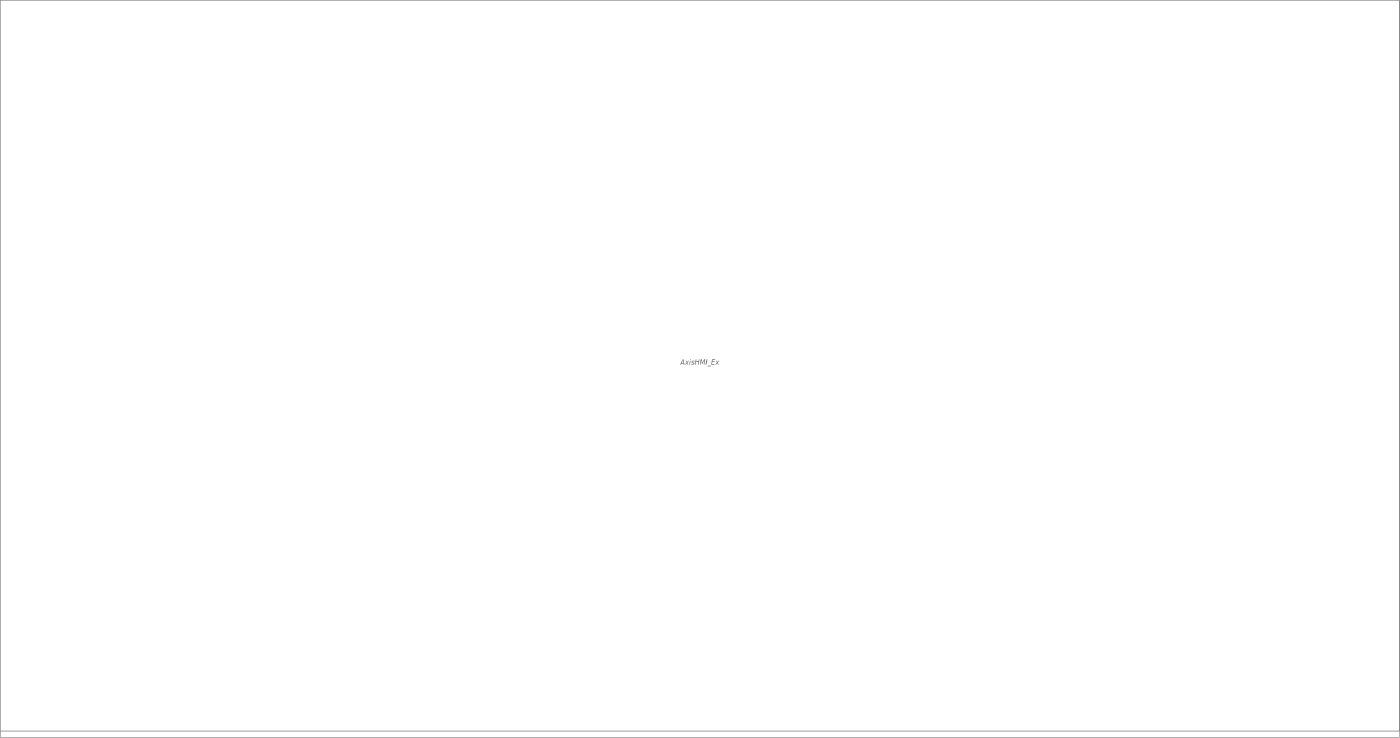
VISUALIZATION visu_working1  // 2048x1080
    TabControl (0,-10 2048x1080)
        shows AxisHMI_Ex(stAxisHMI := GVL.fb_working1.st_mcAxis_lift, mcAxis := GVL.fb_working1.mcAxis_lift, xError := GVL.fb_working1.mcAxis_lift.xError)
        shows AxisHMI_Ex(stAxisHMI := GVL.fb_working1.st_mcAxis_bag, mcAxis := GVL.fb_working1.mcAxis_bag, xError := GVL.fb_working1.mcAxis_bag.xError)
        shows v_io_working1()
        shows AxisHMI_Ex(stAxisHMI := GVL.fb_working.st_mcAxis_vacuun[0], mcAxis := GVL.fb_working.mcAxis_vacuun[0], xError := GVL.fb_working.mcAxis_vacuun[0].xError)
        shows AxisHMI_Ex(stAxisHMI := GVL.fb_working.st_mcAxis_vacuun[1], mcAxis := GVL.fb_working.mcAxis_vacuun[1], xError := GVL.fb_working.mcAxis_vacuun[1].xError)
        shows AxisHMI_Ex(stAxisHMI := GVL.fb_working.st_mcAxis_bagOpen[0], mcAxis := GVL.fb_working.mcAxis_bagOpen[0], xError := GVL.fb_working.mcAxis_bagOpen[0].xError)
        shows AxisHMI_Ex(stAxisHMI := GVL.fb_working.st_mcAxis_bagOpen[1], mcAxis := GVL.fb_working.mcAxis_bagOpen[1], xError := GVL.fb_working.mcAxis_bagOpen[1].xError)
        shows AxisHMI_Ex(stAxisHMI := GVL.fb_working.st_mcAxis_bagOpen[2], mcAxis := GVL.fb_working.mcAxis_bagOpen[2], xError := GVL.fb_working.mcAxis_bagOpen[2].xError)
        shows AxisHMI_Ex(stAxisHMI := GVL.fb_working.st_mcAxis_bagOpen[3], mcAxis := GVL.fb_working.mcAxis_bagOpen[3], xError := GVL.fb_working.mcAxis_bagOpen[3].xError)
        [0]: TabTitle=Lift
        [1]: TabTitle=BagOpen
        [3]: TabTitle=Axis_vacuun_0
        [4]: TabTitle=Axis_vacuun_1
        [5]: TabTitle=Axis_bagOpen_0
        [6]: TabTitle=Axis_bagOpen_1
        [7]: TabTitle=Axis_bagOpen_2
        [8]: TabTitle=Axis_bagOpen_3
        p2837713833: gantrybase.mcAxis[EN_Axis.Z].sAxisName
END_VISUALIZATION

(* stored: Version 1.1.0.1, ProductVersion 3.1.4024.12
   Visu visu_working1: Id {4237067d-ba12-473e-bb87-3d8ec82551ac} *)
